// Mitsubishi GX Works2 project: 사칙연산   PLC: Q02/Q02H

PROGRAM MAIN
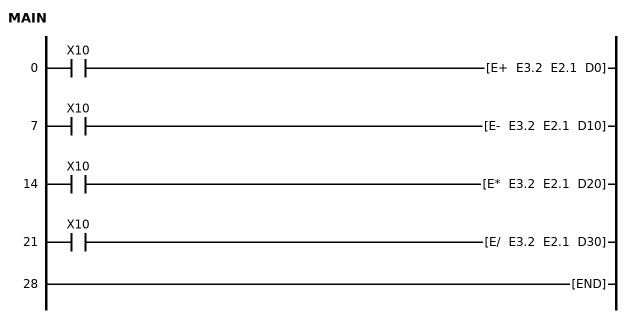
0     LD      X10
      E+      E3.2 E2.1 D0
7     LD      X10
      E-      E3.2 E2.1 D10
14    LD      X10
      E*      E3.2 E2.1 D20
21    LD      X10
      E/      E3.2 E2.1 D30
28    END
END_PROGRAM
